// TIA Portal V21 export
FUNCTION "Gest_LayoutPercorsi" : Void   // FC137, LAD
{ S7_Optimized_Access := 'TRUE' }
// stored: SetENOAutomatically false
   VAR_TEMP
      ProdottoNelTubo : Int;
   END_VAR
   VAR CONSTANT
      Prodotto_Pomodoro : Int := 5;   // Tubo rosso
      Prodotto_AcquaFredda : Int := 1;   // Tubo blu
      Prodotto_Vuoto : Int := 0;   // Tubo grigio chiaro
      Prodotto_Acido : Int := 3;   // Tubazione verde
      Prodotto_Soda : Int := 4;   // Tubazione gialla
      Prodotto_AcquaCalda : Int := 2;   // Tubo grigio
      Prodotto_Vapore : Int := 6;   // Tubazione grigio molto chiaro
      Prodotto_7 : Int := 7;   // Tubazione libea
   END_VAR
   VAR_TEMP   // added for the SCL form of the ladder/FBD networks
      _w1 : Bool;
      _w2 : Bool;
      _w3 : Bool;
   END_VAR
BEGIN

REGION Network 1 (SCL): Prodotto presente nel serbatoio prodotto
   #ProdottoNelTubo := #Prodotto_Vuoto;

   IF "Sequenza".S[K_Sequenza_Produzione].Out.SequenzaAvviata THEN
       #ProdottoNelTubo := #Prodotto_Pomodoro;
       IF "Sequenza".S[K_Sequenza_Produzione].Out.Passo[K_Passo_RisciacquoFineSvuotamento].Attivo THEN
           #ProdottoNelTubo := #Prodotto_AcquaFredda;
       END_IF;
   END_IF;

   IF "Sequenza".S[K_Sequenza_Lavaggio].Out.SequenzaAvviata THEN
       CASE "Sequenza".S[K_Sequenza_Lavaggio].Dati.PassoAttuale OF
           "K_Passo_Acido":
               #ProdottoNelTubo := #Prodotto_Acido;
           "K_Passo_Soda":
               #ProdottoNelTubo := #Prodotto_Soda;
           "K_Passo_Risciacquo":
               #ProdottoNelTubo := #Prodotto_AcquaFredda;
           "K_Passo_RisciacquoAcido":
               #ProdottoNelTubo := #Prodotto_AcquaFredda;
           "K_Passo_RisciacquoSoda":
               #ProdottoNelTubo := #Prodotto_AcquaFredda;
       END_CASE;
   END_IF;

   "LayoutPercorsi".PercorsoDa.SerbatoioProdotto := #ProdottoNelTubo;
END_REGION

REGION Network 2: Prodotto presente nella tubazione dopo drenaggio vasca
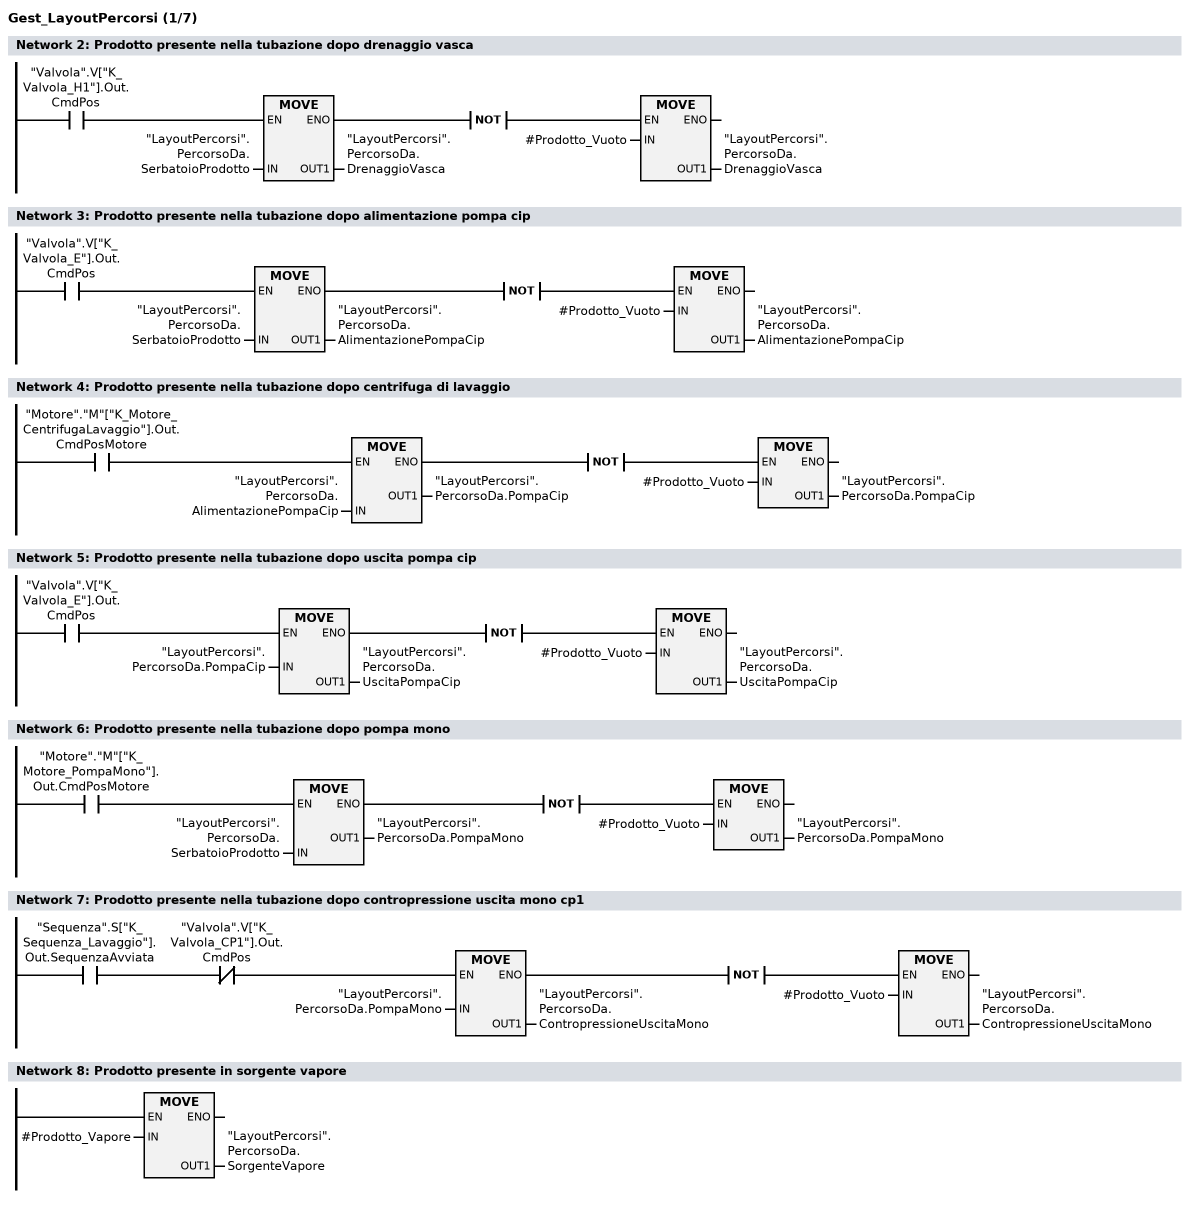
   RUNG wire#powerrail
      Contact( "Valvola".V["K_Valvola_H1"].Out.CmdPos )
      Move(in := "LayoutPercorsi".PercorsoDa.SerbatoioProdotto, out1 => "LayoutPercorsi".PercorsoDa.DrenaggioVasca)
      Not()
      Move(in := #Prodotto_Vuoto, out1 => "LayoutPercorsi".PercorsoDa.DrenaggioVasca)
   END_RUNG
   // the same network as SCL:
   IF "Valvola".V["K_Valvola_H1"].Out.CmdPos THEN
       "LayoutPercorsi".PercorsoDa.DrenaggioVasca := "LayoutPercorsi".PercorsoDa.SerbatoioProdotto;
   END_IF;
   IF NOT "Valvola".V["K_Valvola_H1"].Out.CmdPos THEN
       "LayoutPercorsi".PercorsoDa.DrenaggioVasca := #Prodotto_Vuoto;
   END_IF;
END_REGION

REGION Network 3: Prodotto presente nella tubazione dopo alimentazione pompa cip
   RUNG wire#powerrail
      Contact( "Valvola".V["K_Valvola_E"].Out.CmdPos )
      Move(in := "LayoutPercorsi".PercorsoDa.SerbatoioProdotto, out1 => "LayoutPercorsi".PercorsoDa.AlimentazionePompaCip)
      Not()
      Move(in := #Prodotto_Vuoto, out1 => "LayoutPercorsi".PercorsoDa.AlimentazionePompaCip)
   END_RUNG
   // the same network as SCL:
   IF "Valvola".V["K_Valvola_E"].Out.CmdPos THEN
       "LayoutPercorsi".PercorsoDa.AlimentazionePompaCip := "LayoutPercorsi".PercorsoDa.SerbatoioProdotto;
   END_IF;
   IF NOT "Valvola".V["K_Valvola_E"].Out.CmdPos THEN
       "LayoutPercorsi".PercorsoDa.AlimentazionePompaCip := #Prodotto_Vuoto;
   END_IF;
END_REGION

REGION Network 4: Prodotto presente nella tubazione dopo centrifuga di lavaggio
   RUNG wire#powerrail
      Contact( "Motore"."M"["K_Motore_CentrifugaLavaggio"].Out.CmdPosMotore )
      Move(in := "LayoutPercorsi".PercorsoDa.AlimentazionePompaCip, out1 => "LayoutPercorsi".PercorsoDa.PompaCip)
      Not()
      Move(in := #Prodotto_Vuoto, out1 => "LayoutPercorsi".PercorsoDa.PompaCip)
   END_RUNG
   // the same network as SCL:
   IF "Motore"."M"["K_Motore_CentrifugaLavaggio"].Out.CmdPosMotore THEN
       "LayoutPercorsi".PercorsoDa.PompaCip := "LayoutPercorsi".PercorsoDa.AlimentazionePompaCip;
   END_IF;
   IF NOT "Motore"."M"["K_Motore_CentrifugaLavaggio"].Out.CmdPosMotore THEN
       "LayoutPercorsi".PercorsoDa.PompaCip := #Prodotto_Vuoto;
   END_IF;
END_REGION

REGION Network 5: Prodotto presente nella tubazione dopo uscita pompa cip
   RUNG wire#powerrail
      Contact( "Valvola".V["K_Valvola_E"].Out.CmdPos )
      Move(in := "LayoutPercorsi".PercorsoDa.PompaCip, out1 => "LayoutPercorsi".PercorsoDa.UscitaPompaCip)
      Not()
      Move(in := #Prodotto_Vuoto, out1 => "LayoutPercorsi".PercorsoDa.UscitaPompaCip)
   END_RUNG
   // the same network as SCL:
   IF "Valvola".V["K_Valvola_E"].Out.CmdPos THEN
       "LayoutPercorsi".PercorsoDa.UscitaPompaCip := "LayoutPercorsi".PercorsoDa.PompaCip;
   END_IF;
   IF NOT "Valvola".V["K_Valvola_E"].Out.CmdPos THEN
       "LayoutPercorsi".PercorsoDa.UscitaPompaCip := #Prodotto_Vuoto;
   END_IF;
END_REGION

REGION Network 6: Prodotto presente nella tubazione dopo pompa mono
   RUNG wire#powerrail
      Contact( "Motore"."M"["K_Motore_PompaMono"].Out.CmdPosMotore )
      Move(in := "LayoutPercorsi".PercorsoDa.SerbatoioProdotto, out1 => "LayoutPercorsi".PercorsoDa.PompaMono)
      Not()
      Move(in := #Prodotto_Vuoto, out1 => "LayoutPercorsi".PercorsoDa.PompaMono)
   END_RUNG
   // the same network as SCL:
   IF "Motore"."M"["K_Motore_PompaMono"].Out.CmdPosMotore THEN
       "LayoutPercorsi".PercorsoDa.PompaMono := "LayoutPercorsi".PercorsoDa.SerbatoioProdotto;
   END_IF;
   IF NOT "Motore"."M"["K_Motore_PompaMono"].Out.CmdPosMotore THEN
       "LayoutPercorsi".PercorsoDa.PompaMono := #Prodotto_Vuoto;
   END_IF;
END_REGION

REGION Network 7: Prodotto presente nella tubazione dopo contropressione uscita mono cp1
   RUNG wire#powerrail
      Contact( "Sequenza".S["K_Sequenza_Lavaggio"].Out.SequenzaAvviata )
      I_Contact( "Valvola".V["K_Valvola_CP1"].Out.CmdPos )
      Move(in := "LayoutPercorsi".PercorsoDa.PompaMono, out1 => "LayoutPercorsi".PercorsoDa.ContropressioneUscitaMono)
      Not()
      Move(in := #Prodotto_Vuoto, out1 => "LayoutPercorsi".PercorsoDa.ContropressioneUscitaMono)
   END_RUNG
   // the same network as SCL:
   #_w1 := "Sequenza".S["K_Sequenza_Lavaggio"].Out.SequenzaAvviata AND NOT "Valvola".V["K_Valvola_CP1"].Out.CmdPos;
   IF #_w1 THEN
       "LayoutPercorsi".PercorsoDa.ContropressioneUscitaMono := "LayoutPercorsi".PercorsoDa.PompaMono;
   END_IF;
   IF NOT #_w1 THEN "LayoutPercorsi".PercorsoDa.ContropressioneUscitaMono := #Prodotto_Vuoto; END_IF;
END_REGION

REGION Network 8: Prodotto presente in sorgente vapore
   RUNG wire#powerrail
      Move(in := #Prodotto_Vapore, out1 => "LayoutPercorsi".PercorsoDa.SorgenteVapore)
   END_RUNG
   // the same network as SCL:
   "LayoutPercorsi".PercorsoDa.SorgenteVapore := #Prodotto_Vapore;
END_REGION

REGION Network 9: Prodotto presente nella tubazione dopo Pompa pistoni
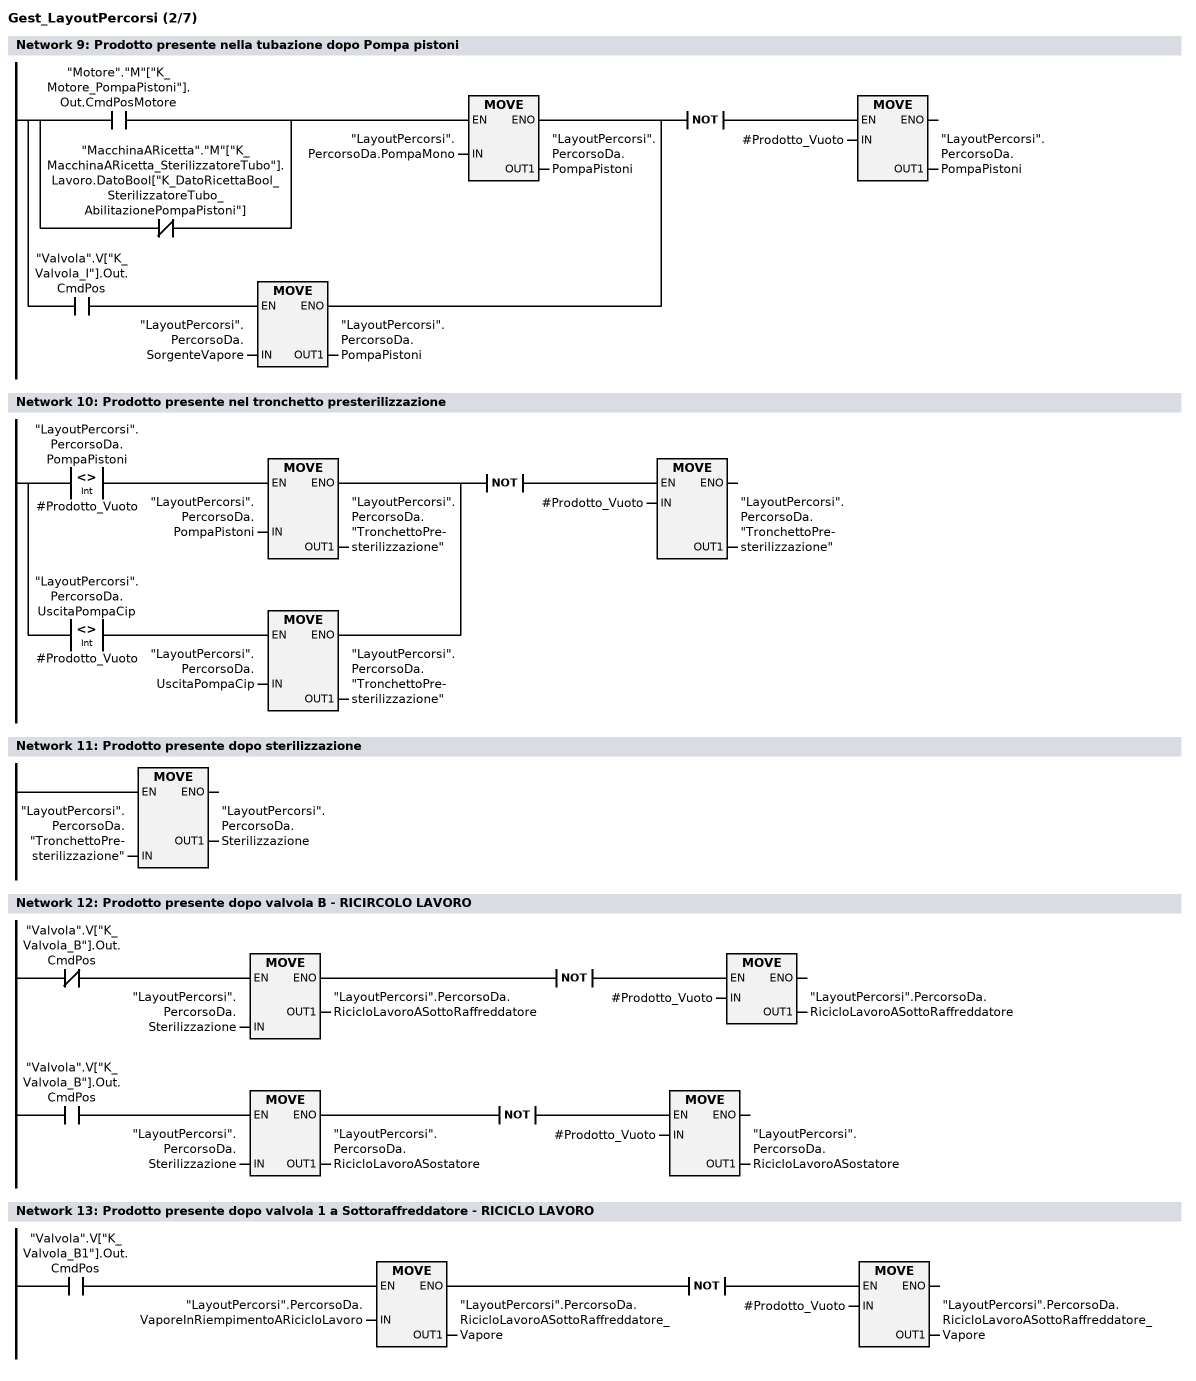
   RUNG wire#powerrail
      Contact( "Motore"."M"["K_Motore_PompaPistoni"].Out.CmdPosMotore )
      wire#w1
      Move(in := "LayoutPercorsi".PercorsoDa.PompaMono, out1 => "LayoutPercorsi".PercorsoDa.PompaPistoni)
      wire#w2
      Not()
      Move(in := #Prodotto_Vuoto, out1 => "LayoutPercorsi".PercorsoDa.PompaPistoni)
   END_RUNG
   RUNG wire#powerrail
      I_Contact( "MacchinaARicetta"."M"["K_MacchinaARicetta_SterilizzatoreTubo"].Lavoro.DatoBool["K_DatoRicettaBool_SterilizzatoreTubo_AbilitazionePompaPistoni"] )
   END_RUNG wire#w1
   RUNG wire#powerrail
      Contact( "Valvola".V["K_Valvola_I"].Out.CmdPos )
      Move(in := "LayoutPercorsi".PercorsoDa.SorgenteVapore, out1 => "LayoutPercorsi".PercorsoDa.PompaPistoni)
   END_RUNG wire#w2
   // the same network as SCL:
   #_w1 := "Motore"."M"["K_Motore_PompaPistoni"].Out.CmdPosMotore OR NOT "MacchinaARicetta"."M"["K_MacchinaARicetta_SterilizzatoreTubo"].Lavoro.DatoBool["K_DatoRicettaBool_SterilizzatoreTubo_AbilitazionePompaPistoni"];
   IF #_w1 THEN "LayoutPercorsi".PercorsoDa.PompaPistoni := "LayoutPercorsi".PercorsoDa.PompaMono; END_IF;
   IF "Valvola".V["K_Valvola_I"].Out.CmdPos THEN
       "LayoutPercorsi".PercorsoDa.PompaPistoni := "LayoutPercorsi".PercorsoDa.SorgenteVapore;
   END_IF;
   IF NOT (#_w1 OR "Valvola".V["K_Valvola_I"].Out.CmdPos) THEN
       "LayoutPercorsi".PercorsoDa.PompaPistoni := #Prodotto_Vuoto;
   END_IF;
END_REGION

REGION Network 10: Prodotto presente nel tronchetto presterilizzazione
   RUNG wire#powerrail
      { S7_Templates := "SrcType := Int" } NE_Contact(in1 := "LayoutPercorsi".PercorsoDa.PompaPistoni, in2 := #Prodotto_Vuoto)
      Move(in := "LayoutPercorsi".PercorsoDa.PompaPistoni, out1 => "LayoutPercorsi".PercorsoDa."TronchettoPre-sterilizzazione")
      wire#w1
      Not()
      Move(in := #Prodotto_Vuoto, out1 => "LayoutPercorsi".PercorsoDa."TronchettoPre-sterilizzazione")
   END_RUNG
   RUNG wire#powerrail
      { S7_Templates := "SrcType := Int" } NE_Contact(in1 := "LayoutPercorsi".PercorsoDa.UscitaPompaCip, in2 := #Prodotto_Vuoto)
      Move(in := "LayoutPercorsi".PercorsoDa.UscitaPompaCip, out1 => "LayoutPercorsi".PercorsoDa."TronchettoPre-sterilizzazione")
   END_RUNG wire#w1
   // the same network as SCL:
   #_w1 := "LayoutPercorsi".PercorsoDa.PompaPistoni <> #Prodotto_Vuoto;
   IF #_w1 THEN
       "LayoutPercorsi".PercorsoDa."TronchettoPre-sterilizzazione" := "LayoutPercorsi".PercorsoDa.PompaPistoni;
   END_IF;
   #_w2 := "LayoutPercorsi".PercorsoDa.UscitaPompaCip <> #Prodotto_Vuoto;
   IF #_w2 THEN
       "LayoutPercorsi".PercorsoDa."TronchettoPre-sterilizzazione" := "LayoutPercorsi".PercorsoDa.UscitaPompaCip;
   END_IF;
   IF NOT (#_w1 OR #_w2) THEN
       "LayoutPercorsi".PercorsoDa."TronchettoPre-sterilizzazione" := #Prodotto_Vuoto;
   END_IF;
END_REGION

REGION Network 11: Prodotto presente dopo sterilizzazione
   RUNG wire#powerrail
      Move(in := "LayoutPercorsi".PercorsoDa."TronchettoPre-sterilizzazione", out1 => "LayoutPercorsi".PercorsoDa.Sterilizzazione)
   END_RUNG
   // the same network as SCL:
   "LayoutPercorsi".PercorsoDa.Sterilizzazione := "LayoutPercorsi".PercorsoDa."TronchettoPre-sterilizzazione";
END_REGION

REGION Network 12: Prodotto presente dopo valvola B - RICIRCOLO LAVORO
   RUNG wire#powerrail
      I_Contact( "Valvola".V["K_Valvola_B"].Out.CmdPos )
      Move(in := "LayoutPercorsi".PercorsoDa.Sterilizzazione, out1 => "LayoutPercorsi".PercorsoDa.RicicloLavoroASottoRaffreddatore)
      Not()
      Move(in := #Prodotto_Vuoto, out1 => "LayoutPercorsi".PercorsoDa.RicicloLavoroASottoRaffreddatore)
   END_RUNG
   RUNG wire#powerrail
      Contact( "Valvola".V["K_Valvola_B"].Out.CmdPos )
      Move(in := "LayoutPercorsi".PercorsoDa.Sterilizzazione, out1 => "LayoutPercorsi".PercorsoDa.RicicloLavoroASostatore)
      Not()
      Move(in := #Prodotto_Vuoto, out1 => "LayoutPercorsi".PercorsoDa.RicicloLavoroASostatore)
   END_RUNG
   // the same network as SCL:
   #_w1 := NOT "Valvola".V["K_Valvola_B"].Out.CmdPos;
   IF #_w1 THEN
       "LayoutPercorsi".PercorsoDa.RicicloLavoroASottoRaffreddatore := "LayoutPercorsi".PercorsoDa.Sterilizzazione;
   END_IF;
   IF NOT #_w1 THEN "LayoutPercorsi".PercorsoDa.RicicloLavoroASottoRaffreddatore := #Prodotto_Vuoto; END_IF;
   IF "Valvola".V["K_Valvola_B"].Out.CmdPos THEN
       "LayoutPercorsi".PercorsoDa.RicicloLavoroASostatore := "LayoutPercorsi".PercorsoDa.Sterilizzazione;
   END_IF;
   IF NOT "Valvola".V["K_Valvola_B"].Out.CmdPos THEN
       "LayoutPercorsi".PercorsoDa.RicicloLavoroASostatore := #Prodotto_Vuoto;
   END_IF;
END_REGION

REGION Network 13: Prodotto presente dopo valvola 1 a Sottoraffreddatore - RICICLO LAVORO
   RUNG wire#powerrail
      Contact( "Valvola".V["K_Valvola_B1"].Out.CmdPos )
      Move(in := "LayoutPercorsi".PercorsoDa.VaporeInRiempimentoARicicloLavoro, out1 => "LayoutPercorsi".PercorsoDa.RicicloLavoroASottoRaffreddatore_Vapore)
      Not()
      Move(in := #Prodotto_Vuoto, out1 => "LayoutPercorsi".PercorsoDa.RicicloLavoroASottoRaffreddatore_Vapore)
   END_RUNG
   // the same network as SCL:
   IF "Valvola".V["K_Valvola_B1"].Out.CmdPos THEN
       "LayoutPercorsi".PercorsoDa.RicicloLavoroASottoRaffreddatore_Vapore := "LayoutPercorsi".PercorsoDa.VaporeInRiempimentoARicicloLavoro;
   END_IF;
   IF NOT "Valvola".V["K_Valvola_B1"].Out.CmdPos THEN
       "LayoutPercorsi".PercorsoDa.RicicloLavoroASottoRaffreddatore_Vapore := #Prodotto_Vuoto;
   END_IF;
END_REGION

REGION Network 14: Prodotto presente dopo ingresso sottoraffreddatore
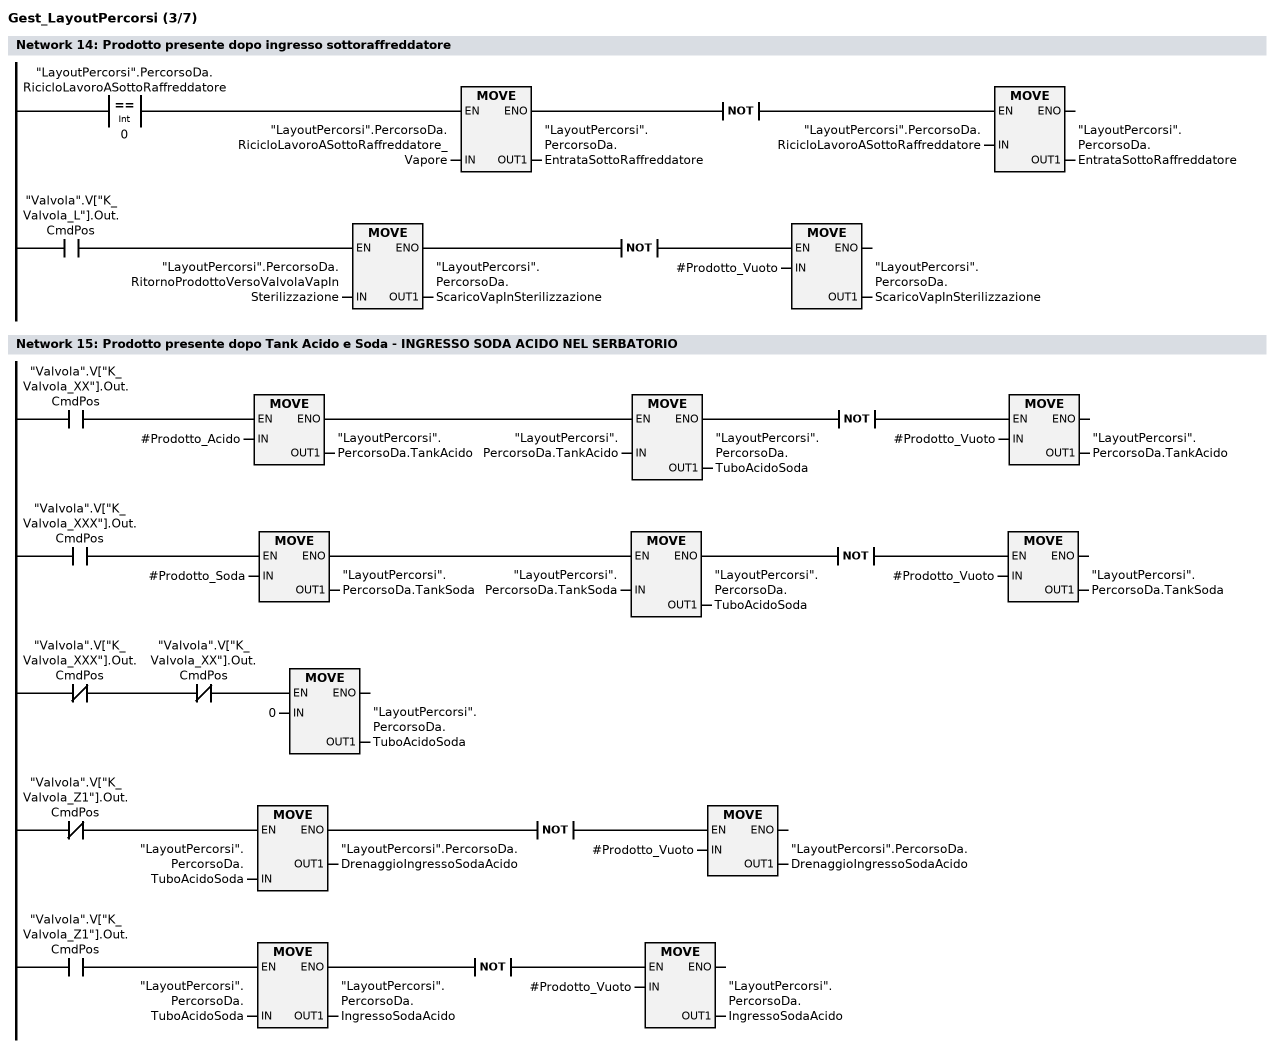
   RUNG wire#powerrail
      { S7_Templates := "SrcType := Int" } EQ_Contact(in1 := "LayoutPercorsi".PercorsoDa.RicicloLavoroASottoRaffreddatore, in2 := 0)
      Move(in := "LayoutPercorsi".PercorsoDa.RicicloLavoroASottoRaffreddatore_Vapore, out1 => "LayoutPercorsi".PercorsoDa.EntrataSottoRaffreddatore)
      Not()
      Move(in := "LayoutPercorsi".PercorsoDa.RicicloLavoroASottoRaffreddatore, out1 => "LayoutPercorsi".PercorsoDa.EntrataSottoRaffreddatore)
   END_RUNG
   RUNG wire#powerrail
      Contact( "Valvola".V["K_Valvola_L"].Out.CmdPos )
      Move(in := "LayoutPercorsi".PercorsoDa.RitornoProdottoVersoValvolaVapInSterilizzazione, out1 => "LayoutPercorsi".PercorsoDa.ScaricoVapInSterilizzazione)
      Not()
      Move(in := #Prodotto_Vuoto, out1 => "LayoutPercorsi".PercorsoDa.ScaricoVapInSterilizzazione)
   END_RUNG
   // the same network as SCL:
   #_w1 := "LayoutPercorsi".PercorsoDa.RicicloLavoroASottoRaffreddatore = 0;
   IF #_w1 THEN
       "LayoutPercorsi".PercorsoDa.EntrataSottoRaffreddatore := "LayoutPercorsi".PercorsoDa.RicicloLavoroASottoRaffreddatore_Vapore;
   END_IF;
   IF NOT #_w1 THEN
       "LayoutPercorsi".PercorsoDa.EntrataSottoRaffreddatore := "LayoutPercorsi".PercorsoDa.RicicloLavoroASottoRaffreddatore;
   END_IF;
   IF "Valvola".V["K_Valvola_L"].Out.CmdPos THEN
       "LayoutPercorsi".PercorsoDa.ScaricoVapInSterilizzazione := "LayoutPercorsi".PercorsoDa.RitornoProdottoVersoValvolaVapInSterilizzazione;
   END_IF;
   IF NOT "Valvola".V["K_Valvola_L"].Out.CmdPos THEN
       "LayoutPercorsi".PercorsoDa.ScaricoVapInSterilizzazione := #Prodotto_Vuoto;
   END_IF;
END_REGION

REGION Network 15: Prodotto presente dopo Tank Acido e Soda - INGRESSO SODA ACIDO NEL SERBATORIO
   RUNG wire#powerrail
      Contact( "Valvola".V["K_Valvola_XX"].Out.CmdPos )
      Move(in := #Prodotto_Acido, out1 => "LayoutPercorsi".PercorsoDa.TankAcido)
      Move(in := "LayoutPercorsi".PercorsoDa.TankAcido, out1 => "LayoutPercorsi".PercorsoDa.TuboAcidoSoda)
      Not()
      Move(in := #Prodotto_Vuoto, out1 => "LayoutPercorsi".PercorsoDa.TankAcido)
   END_RUNG
   RUNG wire#powerrail
      Contact( "Valvola".V["K_Valvola_XXX"].Out.CmdPos )
      Move(in := #Prodotto_Soda, out1 => "LayoutPercorsi".PercorsoDa.TankSoda)
      Move(in := "LayoutPercorsi".PercorsoDa.TankSoda, out1 => "LayoutPercorsi".PercorsoDa.TuboAcidoSoda)
      Not()
      Move(in := #Prodotto_Vuoto, out1 => "LayoutPercorsi".PercorsoDa.TankSoda)
   END_RUNG
   RUNG wire#powerrail
      I_Contact( "Valvola".V["K_Valvola_XXX"].Out.CmdPos )
      I_Contact( "Valvola".V["K_Valvola_XX"].Out.CmdPos )
      Move(in := 0, out1 => "LayoutPercorsi".PercorsoDa.TuboAcidoSoda)
   END_RUNG
   RUNG wire#powerrail
      I_Contact( "Valvola".V["K_Valvola_Z1"].Out.CmdPos )
      Move(in := "LayoutPercorsi".PercorsoDa.TuboAcidoSoda, out1 => "LayoutPercorsi".PercorsoDa.DrenaggioIngressoSodaAcido)
      Not()
      Move(in := #Prodotto_Vuoto, out1 => "LayoutPercorsi".PercorsoDa.DrenaggioIngressoSodaAcido)
   END_RUNG
   RUNG wire#powerrail
      Contact( "Valvola".V["K_Valvola_Z1"].Out.CmdPos )
      Move(in := "LayoutPercorsi".PercorsoDa.TuboAcidoSoda, out1 => "LayoutPercorsi".PercorsoDa.IngressoSodaAcido)
      Not()
      Move(in := #Prodotto_Vuoto, out1 => "LayoutPercorsi".PercorsoDa.IngressoSodaAcido)
   END_RUNG
   // the same network as SCL:
   IF "Valvola".V["K_Valvola_XX"].Out.CmdPos THEN
       "LayoutPercorsi".PercorsoDa.TankAcido := #Prodotto_Acido;
       "LayoutPercorsi".PercorsoDa.TuboAcidoSoda := "LayoutPercorsi".PercorsoDa.TankAcido;
   END_IF;
   IF NOT "Valvola".V["K_Valvola_XX"].Out.CmdPos THEN
       "LayoutPercorsi".PercorsoDa.TankAcido := #Prodotto_Vuoto;
   END_IF;
   IF "Valvola".V["K_Valvola_XXX"].Out.CmdPos THEN
       "LayoutPercorsi".PercorsoDa.TankSoda := #Prodotto_Soda;
       "LayoutPercorsi".PercorsoDa.TuboAcidoSoda := "LayoutPercorsi".PercorsoDa.TankSoda;
   END_IF;
   IF NOT "Valvola".V["K_Valvola_XXX"].Out.CmdPos THEN
       "LayoutPercorsi".PercorsoDa.TankSoda := #Prodotto_Vuoto;
   END_IF;
   IF NOT "Valvola".V["K_Valvola_XXX"].Out.CmdPos AND NOT "Valvola".V["K_Valvola_XX"].Out.CmdPos THEN
       "LayoutPercorsi".PercorsoDa.TuboAcidoSoda := 0;
   END_IF;
   #_w1 := NOT "Valvola".V["K_Valvola_Z1"].Out.CmdPos;
   IF #_w1 THEN
       "LayoutPercorsi".PercorsoDa.DrenaggioIngressoSodaAcido := "LayoutPercorsi".PercorsoDa.TuboAcidoSoda;
   END_IF;
   IF NOT #_w1 THEN "LayoutPercorsi".PercorsoDa.DrenaggioIngressoSodaAcido := #Prodotto_Vuoto; END_IF;
   IF "Valvola".V["K_Valvola_Z1"].Out.CmdPos THEN
       "LayoutPercorsi".PercorsoDa.IngressoSodaAcido := "LayoutPercorsi".PercorsoDa.TuboAcidoSoda;
   END_IF;
   IF NOT "Valvola".V["K_Valvola_Z1"].Out.CmdPos THEN
       "LayoutPercorsi".PercorsoDa.IngressoSodaAcido := #Prodotto_Vuoto;
   END_IF;
END_REGION

REGION Network 16: Prodotto presente dopo sostatore e raffreddatore
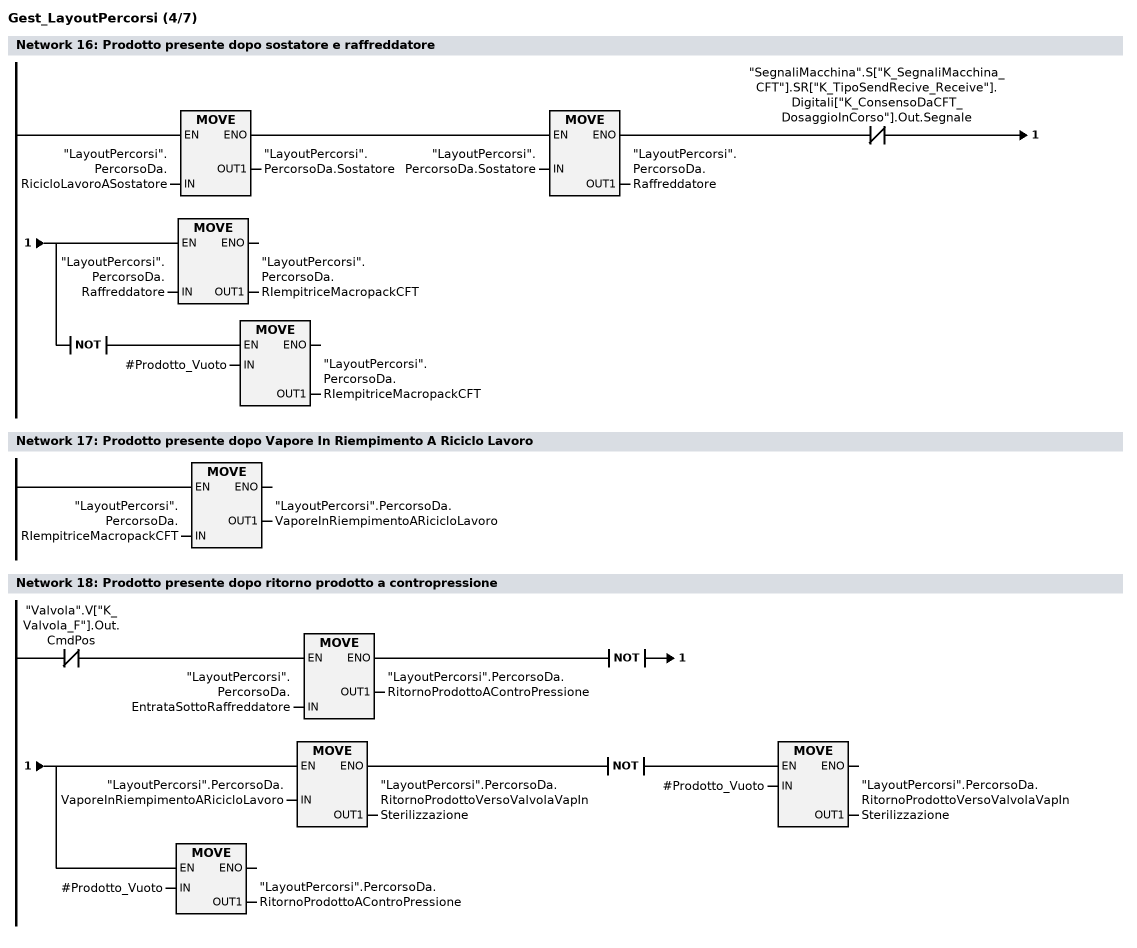
   RUNG wire#powerrail
      Move(in := "LayoutPercorsi".PercorsoDa.RicicloLavoroASostatore, out1 => "LayoutPercorsi".PercorsoDa.Sostatore)
      Move(in := "LayoutPercorsi".PercorsoDa.Sostatore, out1 => "LayoutPercorsi".PercorsoDa.Raffreddatore)
      I_Contact( "SegnaliMacchina".S["K_SegnaliMacchina_CFT"].SR["K_TipoSendRecive_Receive"].Digitali["K_ConsensoDaCFT_DosaggioInCorso"].Out.Segnale )
      wire#w1
      Move(in := "LayoutPercorsi".PercorsoDa.Raffreddatore, out1 => "LayoutPercorsi".PercorsoDa.RIempitriceMacropackCFT)
   END_RUNG
   RUNG wire#w1
      Not()
      Move(in := #Prodotto_Vuoto, out1 => "LayoutPercorsi".PercorsoDa.RIempitriceMacropackCFT)
   END_RUNG
   // the same network as SCL:
   "LayoutPercorsi".PercorsoDa.Sostatore := "LayoutPercorsi".PercorsoDa.RicicloLavoroASostatore;
   "LayoutPercorsi".PercorsoDa.Raffreddatore := "LayoutPercorsi".PercorsoDa.Sostatore;
   #_w1 := NOT "SegnaliMacchina".S["K_SegnaliMacchina_CFT"].SR["K_TipoSendRecive_Receive"].Digitali["K_ConsensoDaCFT_DosaggioInCorso"].Out.Segnale;
   IF #_w1 THEN
       "LayoutPercorsi".PercorsoDa.RIempitriceMacropackCFT := "LayoutPercorsi".PercorsoDa.Raffreddatore;
   END_IF;
   IF NOT #_w1 THEN "LayoutPercorsi".PercorsoDa.RIempitriceMacropackCFT := #Prodotto_Vuoto; END_IF;
END_REGION

REGION Network 17: Prodotto presente dopo Vapore In Riempimento A Riciclo Lavoro
   RUNG wire#powerrail
      Move(in := "LayoutPercorsi".PercorsoDa.RIempitriceMacropackCFT, out1 => "LayoutPercorsi".PercorsoDa.VaporeInRiempimentoARicicloLavoro)
   END_RUNG
   // the same network as SCL:
   "LayoutPercorsi".PercorsoDa.VaporeInRiempimentoARicicloLavoro := "LayoutPercorsi".PercorsoDa.RIempitriceMacropackCFT;
END_REGION

REGION Network 18: Prodotto presente dopo ritorno prodotto a contropressione
   RUNG wire#powerrail
      I_Contact( "Valvola".V["K_Valvola_F"].Out.CmdPos )
      Move(in := "LayoutPercorsi".PercorsoDa.EntrataSottoRaffreddatore, out1 => "LayoutPercorsi".PercorsoDa.RitornoProdottoAControPressione)
      Not()
      wire#w1
      Move(in := "LayoutPercorsi".PercorsoDa.VaporeInRiempimentoARicicloLavoro, out1 => "LayoutPercorsi".PercorsoDa.RitornoProdottoVersoValvolaVapInSterilizzazione)
      Not()
      Move(in := #Prodotto_Vuoto, out1 => "LayoutPercorsi".PercorsoDa.RitornoProdottoVersoValvolaVapInSterilizzazione)
   END_RUNG
   RUNG wire#w1
      Move(in := #Prodotto_Vuoto, out1 => "LayoutPercorsi".PercorsoDa.RitornoProdottoAControPressione)
   END_RUNG
   // the same network as SCL:
   #_w1 := NOT "Valvola".V["K_Valvola_F"].Out.CmdPos;
   IF #_w1 THEN
       "LayoutPercorsi".PercorsoDa.RitornoProdottoAControPressione := "LayoutPercorsi".PercorsoDa.EntrataSottoRaffreddatore;
   END_IF;
   IF NOT #_w1 THEN
       "LayoutPercorsi".PercorsoDa.RitornoProdottoVersoValvolaVapInSterilizzazione := "LayoutPercorsi".PercorsoDa.VaporeInRiempimentoARicicloLavoro;
   END_IF;
   IF NOT (NOT #_w1) THEN
       "LayoutPercorsi".PercorsoDa.RitornoProdottoVersoValvolaVapInSterilizzazione := #Prodotto_Vuoto;
   END_IF;
   IF NOT #_w1 THEN "LayoutPercorsi".PercorsoDa.RitornoProdottoAControPressione := #Prodotto_Vuoto; END_IF;
END_REGION

REGION Network 19: Prodotto presente dopo valvola Contropressione devio acido
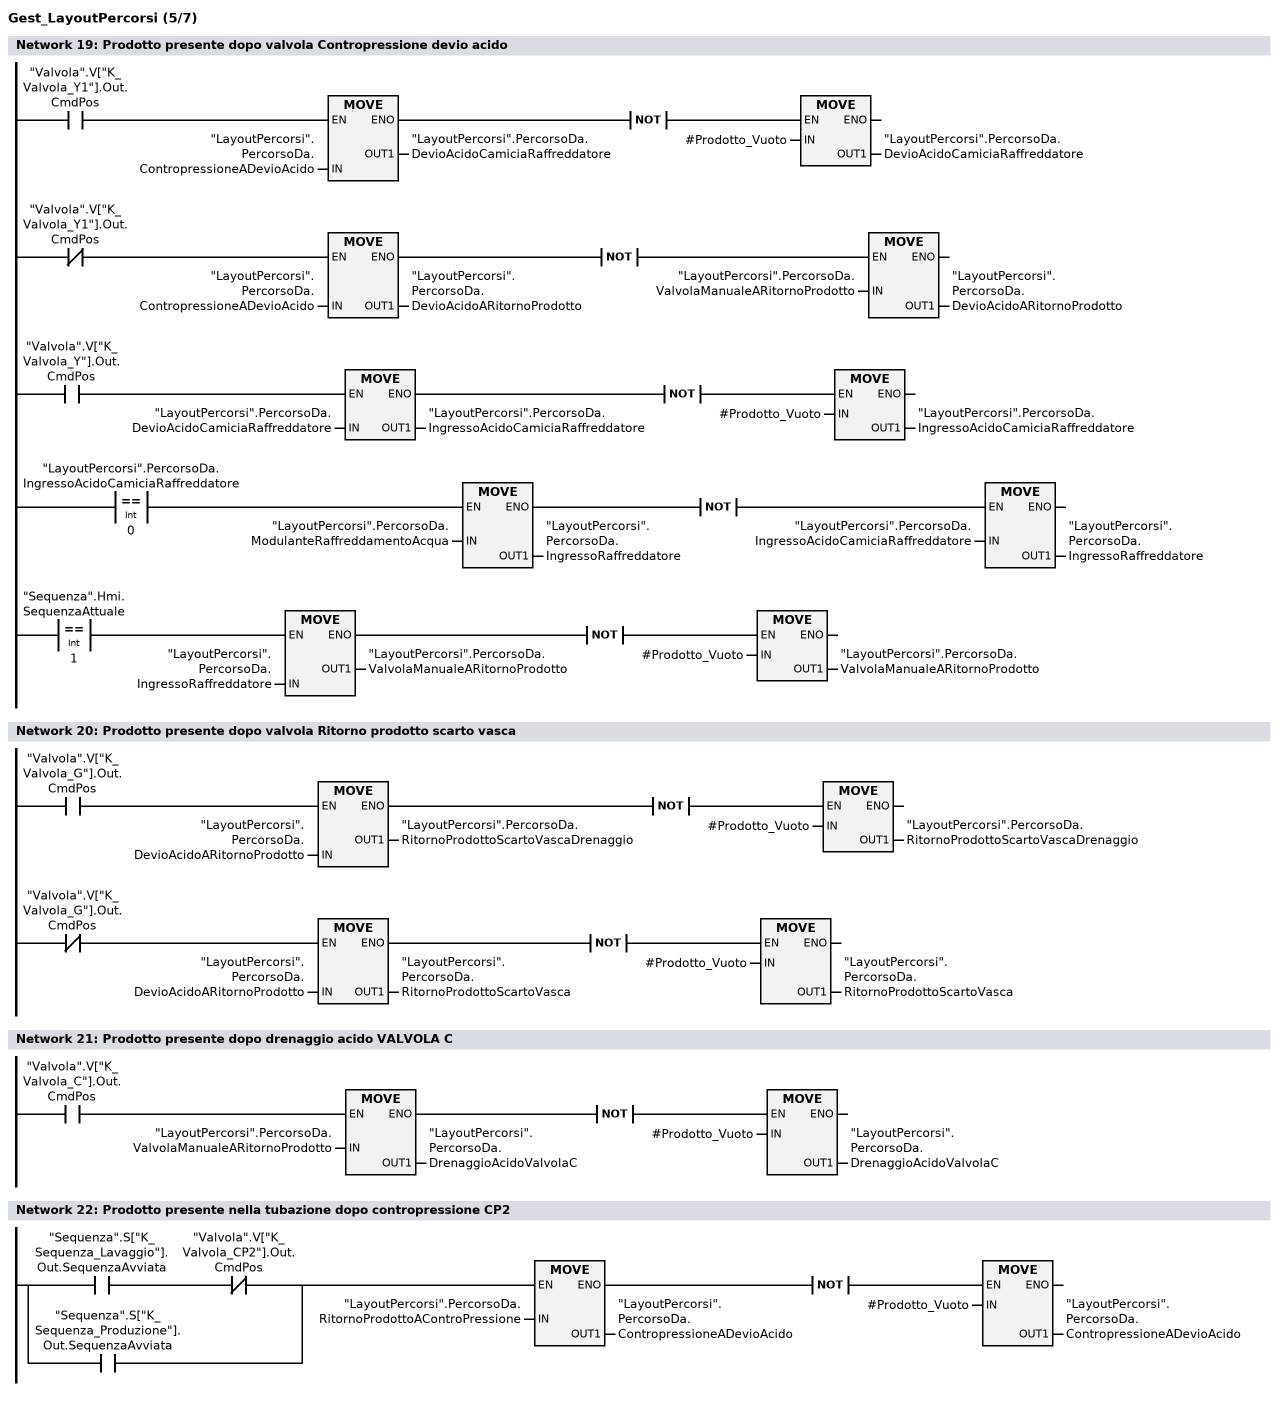
   RUNG wire#powerrail
      Contact( "Valvola".V["K_Valvola_Y1"].Out.CmdPos )
      Move(in := "LayoutPercorsi".PercorsoDa.ContropressioneADevioAcido, out1 => "LayoutPercorsi".PercorsoDa.DevioAcidoCamiciaRaffreddatore)
      Not()
      Move(in := #Prodotto_Vuoto, out1 => "LayoutPercorsi".PercorsoDa.DevioAcidoCamiciaRaffreddatore)
   END_RUNG
   RUNG wire#powerrail
      I_Contact( "Valvola".V["K_Valvola_Y1"].Out.CmdPos )
      Move(in := "LayoutPercorsi".PercorsoDa.ContropressioneADevioAcido, out1 => "LayoutPercorsi".PercorsoDa.DevioAcidoARitornoProdotto)
      Not()
      Move(in := "LayoutPercorsi".PercorsoDa.ValvolaManualeARitornoProdotto, out1 => "LayoutPercorsi".PercorsoDa.DevioAcidoARitornoProdotto)
   END_RUNG
   RUNG wire#powerrail
      Contact( "Valvola".V["K_Valvola_Y"].Out.CmdPos )
      Move(in := "LayoutPercorsi".PercorsoDa.DevioAcidoCamiciaRaffreddatore, out1 => "LayoutPercorsi".PercorsoDa.IngressoAcidoCamiciaRaffreddatore)
      Not()
      Move(in := #Prodotto_Vuoto, out1 => "LayoutPercorsi".PercorsoDa.IngressoAcidoCamiciaRaffreddatore)
   END_RUNG
   RUNG wire#powerrail
      { S7_Templates := "SrcType := Int" } EQ_Contact(in1 := "LayoutPercorsi".PercorsoDa.IngressoAcidoCamiciaRaffreddatore, in2 := 0)
      Move(in := "LayoutPercorsi".PercorsoDa.ModulanteRaffreddamentoAcqua, out1 => "LayoutPercorsi".PercorsoDa.IngressoRaffreddatore)
      Not()
      Move(in := "LayoutPercorsi".PercorsoDa.IngressoAcidoCamiciaRaffreddatore, out1 => "LayoutPercorsi".PercorsoDa.IngressoRaffreddatore)
   END_RUNG
   RUNG wire#powerrail
      { S7_Templates := "SrcType := Int" } EQ_Contact(in1 := "Sequenza".Hmi.SequenzaAttuale, in2 := 1)
      Move(in := "LayoutPercorsi".PercorsoDa.IngressoRaffreddatore, out1 => "LayoutPercorsi".PercorsoDa.ValvolaManualeARitornoProdotto)
      Not()
      Move(in := #Prodotto_Vuoto, out1 => "LayoutPercorsi".PercorsoDa.ValvolaManualeARitornoProdotto)
   END_RUNG
   // the same network as SCL:
   IF "Valvola".V["K_Valvola_Y1"].Out.CmdPos THEN
       "LayoutPercorsi".PercorsoDa.DevioAcidoCamiciaRaffreddatore := "LayoutPercorsi".PercorsoDa.ContropressioneADevioAcido;
   END_IF;
   IF NOT "Valvola".V["K_Valvola_Y1"].Out.CmdPos THEN
       "LayoutPercorsi".PercorsoDa.DevioAcidoCamiciaRaffreddatore := #Prodotto_Vuoto;
   END_IF;
   #_w1 := NOT "Valvola".V["K_Valvola_Y1"].Out.CmdPos;
   IF #_w1 THEN
       "LayoutPercorsi".PercorsoDa.DevioAcidoARitornoProdotto := "LayoutPercorsi".PercorsoDa.ContropressioneADevioAcido;
   END_IF;
   IF NOT #_w1 THEN
       "LayoutPercorsi".PercorsoDa.DevioAcidoARitornoProdotto := "LayoutPercorsi".PercorsoDa.ValvolaManualeARitornoProdotto;
   END_IF;
   IF "Valvola".V["K_Valvola_Y"].Out.CmdPos THEN
       "LayoutPercorsi".PercorsoDa.IngressoAcidoCamiciaRaffreddatore := "LayoutPercorsi".PercorsoDa.DevioAcidoCamiciaRaffreddatore;
   END_IF;
   IF NOT "Valvola".V["K_Valvola_Y"].Out.CmdPos THEN
       "LayoutPercorsi".PercorsoDa.IngressoAcidoCamiciaRaffreddatore := #Prodotto_Vuoto;
   END_IF;
   #_w2 := "LayoutPercorsi".PercorsoDa.IngressoAcidoCamiciaRaffreddatore = 0;
   IF #_w2 THEN
       "LayoutPercorsi".PercorsoDa.IngressoRaffreddatore := "LayoutPercorsi".PercorsoDa.ModulanteRaffreddamentoAcqua;
   END_IF;
   IF NOT #_w2 THEN
       "LayoutPercorsi".PercorsoDa.IngressoRaffreddatore := "LayoutPercorsi".PercorsoDa.IngressoAcidoCamiciaRaffreddatore;
   END_IF;
   #_w3 := "Sequenza".Hmi.SequenzaAttuale = 1;
   IF #_w3 THEN
       "LayoutPercorsi".PercorsoDa.ValvolaManualeARitornoProdotto := "LayoutPercorsi".PercorsoDa.IngressoRaffreddatore;
   END_IF;
   IF NOT #_w3 THEN "LayoutPercorsi".PercorsoDa.ValvolaManualeARitornoProdotto := #Prodotto_Vuoto; END_IF;
END_REGION

REGION Network 20: Prodotto presente dopo valvola Ritorno prodotto scarto vasca
   RUNG wire#powerrail
      Contact( "Valvola".V["K_Valvola_G"].Out.CmdPos )
      Move(in := "LayoutPercorsi".PercorsoDa.DevioAcidoARitornoProdotto, out1 => "LayoutPercorsi".PercorsoDa.RitornoProdottoScartoVascaDrenaggio)
      Not()
      Move(in := #Prodotto_Vuoto, out1 => "LayoutPercorsi".PercorsoDa.RitornoProdottoScartoVascaDrenaggio)
   END_RUNG
   RUNG wire#powerrail
      I_Contact( "Valvola".V["K_Valvola_G"].Out.CmdPos )
      Move(in := "LayoutPercorsi".PercorsoDa.DevioAcidoARitornoProdotto, out1 => "LayoutPercorsi".PercorsoDa.RitornoProdottoScartoVasca)
      Not()
      Move(in := #Prodotto_Vuoto, out1 => "LayoutPercorsi".PercorsoDa.RitornoProdottoScartoVasca)
   END_RUNG
   // the same network as SCL:
   IF "Valvola".V["K_Valvola_G"].Out.CmdPos THEN
       "LayoutPercorsi".PercorsoDa.RitornoProdottoScartoVascaDrenaggio := "LayoutPercorsi".PercorsoDa.DevioAcidoARitornoProdotto;
   END_IF;
   IF NOT "Valvola".V["K_Valvola_G"].Out.CmdPos THEN
       "LayoutPercorsi".PercorsoDa.RitornoProdottoScartoVascaDrenaggio := #Prodotto_Vuoto;
   END_IF;
   #_w1 := NOT "Valvola".V["K_Valvola_G"].Out.CmdPos;
   IF #_w1 THEN
       "LayoutPercorsi".PercorsoDa.RitornoProdottoScartoVasca := "LayoutPercorsi".PercorsoDa.DevioAcidoARitornoProdotto;
   END_IF;
   IF NOT #_w1 THEN "LayoutPercorsi".PercorsoDa.RitornoProdottoScartoVasca := #Prodotto_Vuoto; END_IF;
END_REGION

REGION Network 21: Prodotto presente dopo drenaggio acido VALVOLA C
   RUNG wire#powerrail
      Contact( "Valvola".V["K_Valvola_C"].Out.CmdPos )
      Move(in := "LayoutPercorsi".PercorsoDa.ValvolaManualeARitornoProdotto, out1 => "LayoutPercorsi".PercorsoDa.DrenaggioAcidoValvolaC)
      Not()
      Move(in := #Prodotto_Vuoto, out1 => "LayoutPercorsi".PercorsoDa.DrenaggioAcidoValvolaC)
   END_RUNG
   // the same network as SCL:
   IF "Valvola".V["K_Valvola_C"].Out.CmdPos THEN
       "LayoutPercorsi".PercorsoDa.DrenaggioAcidoValvolaC := "LayoutPercorsi".PercorsoDa.ValvolaManualeARitornoProdotto;
   END_IF;
   IF NOT "Valvola".V["K_Valvola_C"].Out.CmdPos THEN
       "LayoutPercorsi".PercorsoDa.DrenaggioAcidoValvolaC := #Prodotto_Vuoto;
   END_IF;
END_REGION

REGION Network 22: Prodotto presente nella tubazione dopo contropressione CP2
   RUNG wire#powerrail
      Contact( "Sequenza".S["K_Sequenza_Lavaggio"].Out.SequenzaAvviata )
      I_Contact( "Valvola".V["K_Valvola_CP2"].Out.CmdPos )
      wire#w1
      Move(in := "LayoutPercorsi".PercorsoDa.RitornoProdottoAControPressione, out1 => "LayoutPercorsi".PercorsoDa.ContropressioneADevioAcido)
      Not()
      Move(in := #Prodotto_Vuoto, out1 => "LayoutPercorsi".PercorsoDa.ContropressioneADevioAcido)
   END_RUNG
   RUNG wire#powerrail
      Contact( "Sequenza".S["K_Sequenza_Produzione"].Out.SequenzaAvviata )
   END_RUNG wire#w1
   // the same network as SCL:
   #_w1 := ("Sequenza".S["K_Sequenza_Lavaggio"].Out.SequenzaAvviata AND NOT "Valvola".V["K_Valvola_CP2"].Out.CmdPos) OR "Sequenza".S["K_Sequenza_Produzione"].Out.SequenzaAvviata;
   IF #_w1 THEN
       "LayoutPercorsi".PercorsoDa.ContropressioneADevioAcido := "LayoutPercorsi".PercorsoDa.RitornoProdottoAControPressione;
   END_IF;
   IF NOT #_w1 THEN "LayoutPercorsi".PercorsoDa.ContropressioneADevioAcido := #Prodotto_Vuoto; END_IF;
END_REGION

REGION Network 23: Prodotto presente dopo ingresso acqua VALVOLA X
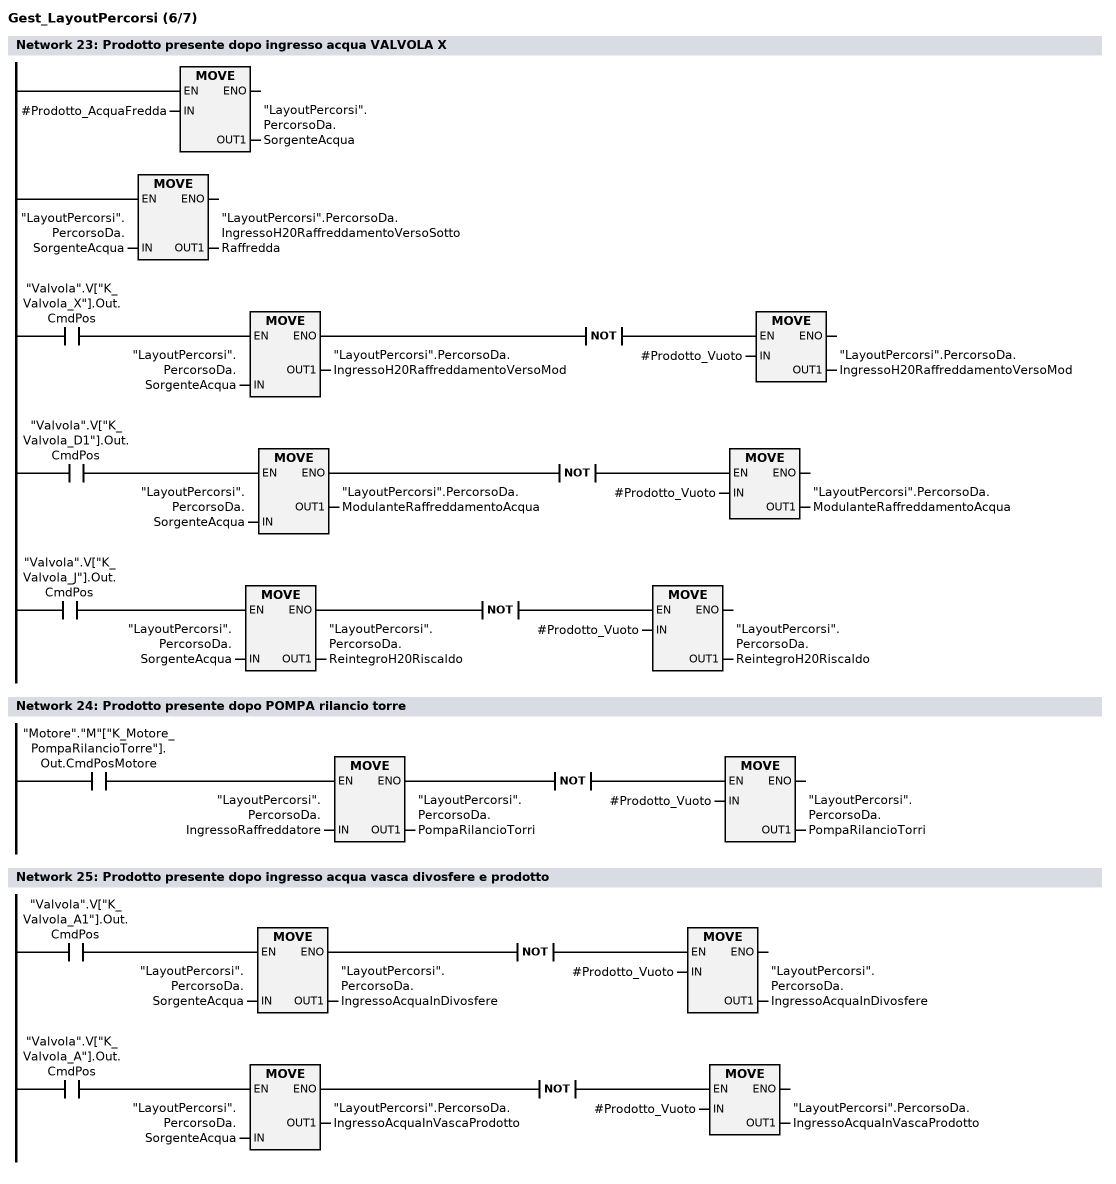
   RUNG wire#powerrail
      Move(in := #Prodotto_AcquaFredda, out1 => "LayoutPercorsi".PercorsoDa.SorgenteAcqua)
   END_RUNG
   RUNG wire#powerrail
      Move(in := "LayoutPercorsi".PercorsoDa.SorgenteAcqua, out1 => "LayoutPercorsi".PercorsoDa.IngressoH20RaffreddamentoVersoSottoRaffredda)
   END_RUNG
   RUNG wire#powerrail
      Contact( "Valvola".V["K_Valvola_X"].Out.CmdPos )
      Move(in := "LayoutPercorsi".PercorsoDa.SorgenteAcqua, out1 => "LayoutPercorsi".PercorsoDa.IngressoH20RaffreddamentoVersoMod)
      Not()
      Move(in := #Prodotto_Vuoto, out1 => "LayoutPercorsi".PercorsoDa.IngressoH20RaffreddamentoVersoMod)
   END_RUNG
   RUNG wire#powerrail
      Contact( "Valvola".V["K_Valvola_D1"].Out.CmdPos )
      Move(in := "LayoutPercorsi".PercorsoDa.SorgenteAcqua, out1 => "LayoutPercorsi".PercorsoDa.ModulanteRaffreddamentoAcqua)
      Not()
      Move(in := #Prodotto_Vuoto, out1 => "LayoutPercorsi".PercorsoDa.ModulanteRaffreddamentoAcqua)
   END_RUNG
   RUNG wire#powerrail
      Contact( "Valvola".V["K_Valvola_J"].Out.CmdPos )
      Move(in := "LayoutPercorsi".PercorsoDa.SorgenteAcqua, out1 => "LayoutPercorsi".PercorsoDa.ReintegroH20Riscaldo)
      Not()
      Move(in := #Prodotto_Vuoto, out1 => "LayoutPercorsi".PercorsoDa.ReintegroH20Riscaldo)
   END_RUNG
   // the same network as SCL:
   "LayoutPercorsi".PercorsoDa.SorgenteAcqua := #Prodotto_AcquaFredda;
   "LayoutPercorsi".PercorsoDa.IngressoH20RaffreddamentoVersoSottoRaffredda := "LayoutPercorsi".PercorsoDa.SorgenteAcqua;
   IF "Valvola".V["K_Valvola_X"].Out.CmdPos THEN
       "LayoutPercorsi".PercorsoDa.IngressoH20RaffreddamentoVersoMod := "LayoutPercorsi".PercorsoDa.SorgenteAcqua;
   END_IF;
   IF NOT "Valvola".V["K_Valvola_X"].Out.CmdPos THEN
       "LayoutPercorsi".PercorsoDa.IngressoH20RaffreddamentoVersoMod := #Prodotto_Vuoto;
   END_IF;
   IF "Valvola".V["K_Valvola_D1"].Out.CmdPos THEN
       "LayoutPercorsi".PercorsoDa.ModulanteRaffreddamentoAcqua := "LayoutPercorsi".PercorsoDa.SorgenteAcqua;
   END_IF;
   IF NOT "Valvola".V["K_Valvola_D1"].Out.CmdPos THEN
       "LayoutPercorsi".PercorsoDa.ModulanteRaffreddamentoAcqua := #Prodotto_Vuoto;
   END_IF;
   IF "Valvola".V["K_Valvola_J"].Out.CmdPos THEN
       "LayoutPercorsi".PercorsoDa.ReintegroH20Riscaldo := "LayoutPercorsi".PercorsoDa.SorgenteAcqua;
   END_IF;
   IF NOT "Valvola".V["K_Valvola_J"].Out.CmdPos THEN
       "LayoutPercorsi".PercorsoDa.ReintegroH20Riscaldo := #Prodotto_Vuoto;
   END_IF;
END_REGION

REGION Network 24: Prodotto presente dopo POMPA rilancio torre
   RUNG wire#powerrail
      Contact( "Motore"."M"["K_Motore_PompaRilancioTorre"].Out.CmdPosMotore )
      Move(in := "LayoutPercorsi".PercorsoDa.IngressoRaffreddatore, out1 => "LayoutPercorsi".PercorsoDa.PompaRilancioTorri)
      Not()
      Move(in := #Prodotto_Vuoto, out1 => "LayoutPercorsi".PercorsoDa.PompaRilancioTorri)
   END_RUNG
   // the same network as SCL:
   IF "Motore"."M"["K_Motore_PompaRilancioTorre"].Out.CmdPosMotore THEN
       "LayoutPercorsi".PercorsoDa.PompaRilancioTorri := "LayoutPercorsi".PercorsoDa.IngressoRaffreddatore;
   END_IF;
   IF NOT "Motore"."M"["K_Motore_PompaRilancioTorre"].Out.CmdPosMotore THEN
       "LayoutPercorsi".PercorsoDa.PompaRilancioTorri := #Prodotto_Vuoto;
   END_IF;
END_REGION

REGION Network 25: Prodotto presente dopo ingresso acqua vasca divosfere e prodotto
   RUNG wire#powerrail
      Contact( "Valvola".V["K_Valvola_A1"].Out.CmdPos )
      Move(in := "LayoutPercorsi".PercorsoDa.SorgenteAcqua, out1 => "LayoutPercorsi".PercorsoDa.IngressoAcquaInDivosfere)
      Not()
      Move(in := #Prodotto_Vuoto, out1 => "LayoutPercorsi".PercorsoDa.IngressoAcquaInDivosfere)
   END_RUNG
   RUNG wire#powerrail
      Contact( "Valvola".V["K_Valvola_A"].Out.CmdPos )
      Move(in := "LayoutPercorsi".PercorsoDa.SorgenteAcqua, out1 => "LayoutPercorsi".PercorsoDa.IngressoAcquaInVascaProdotto)
      Not()
      Move(in := #Prodotto_Vuoto, out1 => "LayoutPercorsi".PercorsoDa.IngressoAcquaInVascaProdotto)
   END_RUNG
   // the same network as SCL:
   IF "Valvola".V["K_Valvola_A1"].Out.CmdPos THEN
       "LayoutPercorsi".PercorsoDa.IngressoAcquaInDivosfere := "LayoutPercorsi".PercorsoDa.SorgenteAcqua;
   END_IF;
   IF NOT "Valvola".V["K_Valvola_A1"].Out.CmdPos THEN
       "LayoutPercorsi".PercorsoDa.IngressoAcquaInDivosfere := #Prodotto_Vuoto;
   END_IF;
   IF "Valvola".V["K_Valvola_A"].Out.CmdPos THEN
       "LayoutPercorsi".PercorsoDa.IngressoAcquaInVascaProdotto := "LayoutPercorsi".PercorsoDa.SorgenteAcqua;
   END_IF;
   IF NOT "Valvola".V["K_Valvola_A"].Out.CmdPos THEN
       "LayoutPercorsi".PercorsoDa.IngressoAcquaInVascaProdotto := #Prodotto_Vuoto;
   END_IF;
END_REGION

REGION Network 26: Prodotto presente dopo QCI
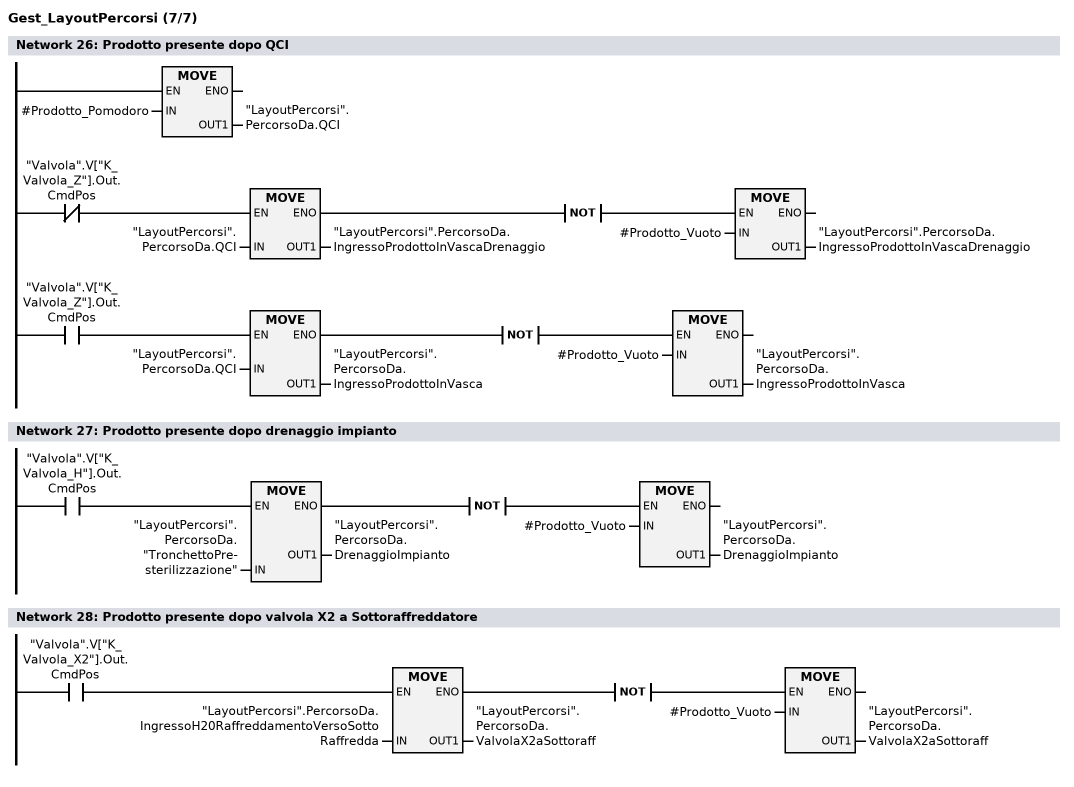
   RUNG wire#powerrail
      Move(in := #Prodotto_Pomodoro, out1 => "LayoutPercorsi".PercorsoDa.QCI)
   END_RUNG
   RUNG wire#powerrail
      I_Contact( "Valvola".V["K_Valvola_Z"].Out.CmdPos )
      Move(in := "LayoutPercorsi".PercorsoDa.QCI, out1 => "LayoutPercorsi".PercorsoDa.IngressoProdottoInVascaDrenaggio)
      Not()
      Move(in := #Prodotto_Vuoto, out1 => "LayoutPercorsi".PercorsoDa.IngressoProdottoInVascaDrenaggio)
   END_RUNG
   RUNG wire#powerrail
      Contact( "Valvola".V["K_Valvola_Z"].Out.CmdPos )
      Move(in := "LayoutPercorsi".PercorsoDa.QCI, out1 => "LayoutPercorsi".PercorsoDa.IngressoProdottoInVasca)
      Not()
      Move(in := #Prodotto_Vuoto, out1 => "LayoutPercorsi".PercorsoDa.IngressoProdottoInVasca)
   END_RUNG
   // the same network as SCL:
   "LayoutPercorsi".PercorsoDa.QCI := #Prodotto_Pomodoro;
   #_w1 := NOT "Valvola".V["K_Valvola_Z"].Out.CmdPos;
   IF #_w1 THEN
       "LayoutPercorsi".PercorsoDa.IngressoProdottoInVascaDrenaggio := "LayoutPercorsi".PercorsoDa.QCI;
   END_IF;
   IF NOT #_w1 THEN "LayoutPercorsi".PercorsoDa.IngressoProdottoInVascaDrenaggio := #Prodotto_Vuoto; END_IF;
   IF "Valvola".V["K_Valvola_Z"].Out.CmdPos THEN
       "LayoutPercorsi".PercorsoDa.IngressoProdottoInVasca := "LayoutPercorsi".PercorsoDa.QCI;
   END_IF;
   IF NOT "Valvola".V["K_Valvola_Z"].Out.CmdPos THEN
       "LayoutPercorsi".PercorsoDa.IngressoProdottoInVasca := #Prodotto_Vuoto;
   END_IF;
END_REGION

REGION Network 27: Prodotto presente dopo drenaggio impianto
   RUNG wire#powerrail
      Contact( "Valvola".V["K_Valvola_H"].Out.CmdPos )
      Move(in := "LayoutPercorsi".PercorsoDa."TronchettoPre-sterilizzazione", out1 => "LayoutPercorsi".PercorsoDa.DrenaggioImpianto)
      Not()
      Move(in := #Prodotto_Vuoto, out1 => "LayoutPercorsi".PercorsoDa.DrenaggioImpianto)
   END_RUNG
   // the same network as SCL:
   IF "Valvola".V["K_Valvola_H"].Out.CmdPos THEN
       "LayoutPercorsi".PercorsoDa.DrenaggioImpianto := "LayoutPercorsi".PercorsoDa."TronchettoPre-sterilizzazione";
   END_IF;
   IF NOT "Valvola".V["K_Valvola_H"].Out.CmdPos THEN
       "LayoutPercorsi".PercorsoDa.DrenaggioImpianto := #Prodotto_Vuoto;
   END_IF;
END_REGION

REGION Network 28: Prodotto presente dopo valvola X2 a Sottoraffreddatore
   RUNG wire#powerrail
      Contact( "Valvola".V["K_Valvola_X2"].Out.CmdPos )
      Move(in := "LayoutPercorsi".PercorsoDa.IngressoH20RaffreddamentoVersoSottoRaffredda, out1 => "LayoutPercorsi".PercorsoDa.ValvolaX2aSottoraff)
      Not()
      Move(in := #Prodotto_Vuoto, out1 => "LayoutPercorsi".PercorsoDa.ValvolaX2aSottoraff)
   END_RUNG
   // the same network as SCL:
   IF "Valvola".V["K_Valvola_X2"].Out.CmdPos THEN
       "LayoutPercorsi".PercorsoDa.ValvolaX2aSottoraff := "LayoutPercorsi".PercorsoDa.IngressoH20RaffreddamentoVersoSottoRaffredda;
   END_IF;
   IF NOT "Valvola".V["K_Valvola_X2"].Out.CmdPos THEN
       "LayoutPercorsi".PercorsoDa.ValvolaX2aSottoraff := #Prodotto_Vuoto;
   END_IF;
END_REGION

REGION Network 29 (SCL): Visbilità della pompa pistoni
   "LayoutPercorsi".Visibilità.PompaPistoni := "MacchinaARicetta".M[K_MacchinaARicetta_SterilizzatoreTubo].Lavoro.DatoBool[K_DatoRicettaBool_SterilizzatoreTubo_AbilitazionePompaPistoni];
END_REGION
END_FUNCTION
